PROGRAM prgCS1
VAR
	fbAlfen1					: FB_ECS_Alfen_NG9xx_Platform;						//{#lynus.ag#()}
	fbAlfen2					: FB_ECS_Alfen_NG9xx_Platform;						//{#lynus.ag#()}
	fbAlfen3					: FB_ECS_Alfen_NG9xx_Platform;						//{#lynus.ag#()}
	fbAlfen4					: FB_ECS_Alfen_NG9xx_Platform;						//{#lynus.ag#()}
	fbAlfen5					: FB_ECS_Alfen_NG9xx_Platform;						//{#lynus.ag#()}
	fbAlfen6					: FB_ECS_Alfen_NG9xx_Platform;						//{#lynus.ag#()}
	fbAlfen7					: FB_ECS_Alfen_NG9xx_Platform;						//{#lynus.ag#()}
	fbAlfen8					: FB_ECS_Alfen_NG9xx_Platform;						//{#lynus.ag#()}
	fbAlfen9					: FB_ECS_Alfen_NG9xx_Platform;						//{#lynus.ag#()}
	fbAlfen10					: FB_ECS_Alfen_NG9xx_Platform;						//{#lynus.ag#()}
	fbApliT_1					: FB_ECS_Alpitronic_Hypercharger;					//{#lynus.ag#()}
	fbApliT_2					: FB_ECS_Alpitronic_Hypercharger;					//{#lynus.ag#()}
	
	bSManualyOn_UV1_1			: BOOL;												//{#lynus.ag#()}
	bySManualyTargetPowerUV1_1	: BYTE;												//{#lynus.ag#()}
	byErrorWarningUV1_1			: BYTE;												//{#lynus.ag#()}
	rChargingTimeInMinUV1_1		: REAL;												//{#lynus.ag#()}
	lrPowerUV1_1				: LREAL;											//{#lynus.ag#()}
	wStateUV1_1					: WORD;												//{#lynus.ag#()}
	lrEnergySessionUV1_1		: LREAL;											//{#lynus.ag#()}
	lrTotalEnergyUV1_1			: LREAL;											//{#lynus.ag#()}
	
	bSManualyOn_UV1_2			: BOOL;												//{#lynus.ag#()}
	bySManualyTargetPowerUV1_2	: BYTE;												//{#lynus.ag#()}
	byErrorWarningUV1_2			: BYTE;												//{#lynus.ag#()}
	rChargingTimeInMinUV1_2		: REAL;												//{#lynus.ag#()}
	lrPowerUV1_2				: LREAL;											//{#lynus.ag#()}
	wStateUV1_2					: WORD;												//{#lynus.ag#()}
	lrEnergySessionUV1_2		: LREAL;											//{#lynus.ag#()}
	lrTotalEnergyUV1_2			: LREAL;											//{#lynus.ag#()}
	
	bSManualyOn_UV1_3			: BOOL;												//{#lynus.ag#()}
	bySManualyTargetPowerUV1_3	: BYTE;												//{#lynus.ag#()}
	byErrorWarningUV1_3			: BYTE;												//{#lynus.ag#()}
	rChargingTimeInMinUV1_3		: REAL;												//{#lynus.ag#()}
	lrPowerUV1_3				: LREAL;											//{#lynus.ag#()}
	wStateUV1_3					: WORD;												//{#lynus.ag#()}
	lrEnergySessionUV1_3		: LREAL;											//{#lynus.ag#()}
	lrTotalEnergyUV1_3			: LREAL;											//{#lynus.ag#()}
	
	bSManualyOn_UV1_4			: BOOL;												//{#lynus.ag#()}
	bySManualyTargetPowerUV1_4	: BYTE;												//{#lynus.ag#()}
	byErrorWarningUV1_4			: BYTE;												//{#lynus.ag#()}
	rChargingTimeInMinUV1_4		: REAL;												//{#lynus.ag#()}
	lrPowerUV1_4				: LREAL;											//{#lynus.ag#()}
	wStateUV1_4					: WORD;												//{#lynus.ag#()}
	lrEnergySessionUV1_4		: LREAL;											//{#lynus.ag#()}
	lrTotalEnergyUV1_4			: LREAL;											//{#lynus.ag#()}
	
	bSManualyOn_UV1_5			: BOOL;												//{#lynus.ag#()}
	bySManualyTargetPowerUV1_5	: BYTE;												//{#lynus.ag#()}
	byErrorWarningUV1_5			: BYTE;												//{#lynus.ag#()}
	rChargingTimeInMinUV1_5		: REAL;												//{#lynus.ag#()}
	lrPowerUV1_5				: LREAL;											//{#lynus.ag#()}
	wStateUV1_5					: WORD;												//{#lynus.ag#()}
	lrEnergySessionUV1_5		: LREAL;											//{#lynus.ag#()}
	lrTotalEnergyUV1_5			: LREAL;											//{#lynus.ag#()}
	
	bSManualyOn_UV1_6			: BOOL;												//{#lynus.ag#()}
	bySManualyTargetPowerUV1_6	: BYTE;												//{#lynus.ag#()}
	byErrorWarningUV1_6			: BYTE;												//{#lynus.ag#()}
	rChargingTimeInMinUV1_6		: REAL;												//{#lynus.ag#()}
	lrPowerUV1_6				: LREAL;											//{#lynus.ag#()}
	wStateUV1_6					: WORD;												//{#lynus.ag#()}
	lrEnergySessionUV1_6		: LREAL;											//{#lynus.ag#()}
	lrTotalEnergyUV1_6			: LREAL;											//{#lynus.ag#()}
	
	bSManualyOn_UV1_7			: BOOL;												//{#lynus.ag#()}
	bySManualyTargetPowerUV1_7	: BYTE;												//{#lynus.ag#()}
	byErrorWarningUV1_7			: BYTE;												//{#lynus.ag#()}
	rChargingTimeInMinUV1_7		: REAL;												//{#lynus.ag#()}
	lrPowerUV1_7				: LREAL;											//{#lynus.ag#()}
	wStateUV1_7					: WORD;												//{#lynus.ag#()}
	lrEnergySessionUV1_7		: LREAL;											//{#lynus.ag#()}
	lrTotalEnergyUV1_7			: LREAL;											//{#lynus.ag#()}
	
	bSManualyOn_UV1_8			: BOOL;												//{#lynus.ag#()}
	bySManualyTargetPowerUV1_8	: BYTE;												//{#lynus.ag#()}
	byErrorWarningUV1_8			: BYTE;												//{#lynus.ag#()}
	rChargingTimeInMinUV1_8		: REAL;												//{#lynus.ag#()}
	lrPowerUV1_8				: LREAL;											//{#lynus.ag#()}
	wStateUV1_8					: WORD;												//{#lynus.ag#()}
	lrEnergySessionUV1_8		: LREAL;											//{#lynus.ag#()}
	lrTotalEnergyUV1_8			: LREAL;											//{#lynus.ag#()}
	
	bSManualyOn_UV1_9			: BOOL;												//{#lynus.ag#()}
	bySManualyTargetPowerUV1_9	: BYTE;												//{#lynus.ag#()}
	byErrorWarningUV1_9			: BYTE;												//{#lynus.ag#()}
	rChargingTimeInMinUV1_9		: REAL;												//{#lynus.ag#()}
	lrPowerUV1_9				: LREAL;											//{#lynus.ag#()}
	wStateUV1_9					: WORD;												//{#lynus.ag#()}
	lrEnergySessionUV1_9		: LREAL;											//{#lynus.ag#()}
	lrTotalEnergyUV1_9			: LREAL;											//{#lynus.ag#()}
	
	bSManualyOn_UV1_10			: BOOL;												//{#lynus.ag#()}
	bySManualyTargetPowerUV1_10	: BYTE;												//{#lynus.ag#()}
	byErrorWarningUV1_10		: BYTE;												//{#lynus.ag#()}
	rChargingTimeInMinUV1_10	: REAL;												//{#lynus.ag#()}
	lrPowerUV1_10				: LREAL;											//{#lynus.ag#()}
	wStateUV1_10				: WORD;												//{#lynus.ag#()}
	lrEnergySessionUV1_10		: LREAL;											//{#lynus.ag#()}
	lrTotalEnergyUV1_10			: LREAL;											//{#lynus.ag#()}
	
	bSManualyOn_DC_1			: BOOL;												//{#lynus.ag#()}
	bySManualyTargetPowerDC_1	: BYTE;												//{#lynus.ag#()}
	byErrorWarningDC_1			: BYTE;												//{#lynus.ag#()}
	lrPowerTotalDC1				: LREAL;											//{#lynus.ag#()}
	lrPowerDC1_S1				: LREAL;											//{#lynus.ag#()}
	lrPowerDC1_S2				: LREAL;											//{#lynus.ag#()}
	rChargingTimeInMinDC1_S1	: REAL;												//{#lynus.ag#()}
	rChargingTimeInMinDC1_S2	: REAL;												//{#lynus.ag#()}
	dwSOCCarDC1_S1				: DWORD;											//{#lynus.ag#()}
	dwSOCCarDC1_S2				: DWORD;											//{#lynus.ag#()}
	wStateDC1_S1				: WORD;												//{#lynus.ag#()}
	wStateDC1_S2				: WORD;												//{#lynus.ag#()}
	lrEnergySessionDC1_S1		: LREAL;											//{#lynus.ag#()}
	lrEnergySessionDC1_S2		: LREAL;											//{#lynus.ag#()}
	lrTotalEnergyDC1			: LREAL;											//{#lynus.ag#()}
	
	bSManualyOn_DC_2			: BOOL;												//{#lynus.ag#()}
	bySManualyTargetPowerDC_2	: BYTE;												//{#lynus.ag#()}
	byErrorWarningDC_2			: BYTE;												//{#lynus.ag#()}
	lrPowerTotalDC2				: LREAL;											//{#lynus.ag#()}
	lrPowerDC2_S1				: LREAL;											//{#lynus.ag#()}
	lrPowerDC2_S2				: LREAL;											//{#lynus.ag#()}
	rChargingTimeInMinDC2_S1	: REAL;												//{#lynus.ag#()}
	rChargingTimeInMinDC2_S2	: REAL;												//{#lynus.ag#()}
	dwSOCCarDC2_S1				: DWORD;											//{#lynus.ag#()}
	dwSOCCarDC2_S2				: DWORD;											//{#lynus.ag#()}
	wStateDC2_S1				: WORD;												//{#lynus.ag#()}
	wStateDC2_S2				: WORD;												//{#lynus.ag#()}
	lrEnergySessionDC2_S1		: LREAL;											//{#lynus.ag#()}
	lrEnergySessionDC2_S2		: LREAL;											//{#lynus.ag#()}
	lrTotalEnergyDC2			: LREAL;											//{#lynus.ag#()}
END_VAR
VAR PERSISTENT
	bManualyOnUV1_1				: BOOL;												//{#lynus.ag#()}
	byManualyTargetPowerUV1_1	: BYTE;												//{#lynus.ag#()}
	
	bManualyOnUV1_2				: BOOL;												//{#lynus.ag#()}
	byManualyTargetPowerUV1_2	: BYTE;												//{#lynus.ag#()}
	
	bManualyOnUV1_3				: BOOL;												//{#lynus.ag#()}
	byManualyTargetPowerUV1_3	: BYTE;												//{#lynus.ag#()}
	
	bManualyOnUV1_4				: BOOL;												//{#lynus.ag#()}
	byManualyTargetPowerUV1_4	: BYTE;												//{#lynus.ag#()}
	
	bManualyOnUV1_5				: BOOL;												//{#lynus.ag#()}
	byManualyTargetPowerUV1_5	: BYTE;												//{#lynus.ag#()}
	
	bManualyOnUV1_6				: BOOL;												//{#lynus.ag#()}
	byManualyTargetPowerUV1_6	: BYTE;												//{#lynus.ag#()}
	
	bManualyOnUV1_7				: BOOL;												//{#lynus.ag#()}
	byManualyTargetPowerUV1_7	: BYTE;												//{#lynus.ag#()}
	
	bManualyOnUV1_8				: BOOL;												//{#lynus.ag#()}
	byManualyTargetPowerUV1_8	: BYTE;												//{#lynus.ag#()}
	
	bManualyOnUV1_9				: BOOL;												//{#lynus.ag#()}
	byManualyTargetPowerUV1_9	: BYTE;												//{#lynus.ag#()}
	
	bManualyOnUV1_10			: BOOL;												//{#lynus.ag#()}
	byManualyTargetPowerUV1_10	: BYTE;												//{#lynus.ag#()}
	
	bManualyOnDC_1				: BOOL;												//{#lynus.ag#()}
	byManualyTargetPowerDC_1	: BYTE;												//{#lynus.ag#()}
	
	bManualyOnDC_2				: BOOL;												//{#lynus.ag#()}
	byManualyTargetPowerDC_2	: BYTE;												//{#lynus.ag#()}
END_VAR

(*---------------------------------------------CS1-----------------------------------------------------------*)

//Manual Power
fbAlfen1.stSetupECS.bManualyOn := bManualyOnUV1_1;
	fbAlfen1.stSetupECS.byManualyTargetPower := byManualyTargetPowerUV1_1;

fbAlfen1(
	bEnable:= , 
	bPowerDataInvers:= , 
	byElectricFuseLine:= , 
	byUnitID_Socket1:= 1, 
	byUnitID_Socket2:= , 
	byNumberOfSockets:= 1, 
	byNumberOfConnectionWire:= 1, 
	diNrOfEMS_IN:= prgEMS.fbEMS.diNrOfEMS_OUT, 
	diNrOfEM_IN_CS:= , 
	sIPAdress:= '192.168.1.123', 
	stSetupECS:= , 
	stDataECS=> , 
	diNrOfECS_OUT=> );

bSManualyOn_UV1_1 := fbAlfen1.stDataECS.bSManualyOn;
	bySManualyTargetPowerUV1_1 := fbAlfen1.stDataECS.bySManualyTargetPower;
		byErrorWarningUV1_1 := fbAlfen1.stDataECS.byErrorWarning;	
			rChargingTimeInMinUV1_1 := fbAlfen1.stDataECS.arrChargingTimeInMin[1];
				lrPowerUV1_1 := fbAlfen1.stDataECS.lrTotalPower;	
					wStateUV1_1 := fbAlfen1.stDataECS.arrSocketStateECS[1];
						lrEnergySessionUV1_1 := fbAlfen1.stDataECS.arrSocketEnergySession[1];
							lrTotalEnergyUV1_1 := fbAlfen1.stDataECS.lrTotalCounterEnergy_Consumption;		
	
(*---------------------------------------------CS2-----------------------------------------------------------*)
	
//Manual Power
fbAlfen2.stSetupECS.bManualyOn := bManualyOnUV1_2;
	fbAlfen2.stSetupECS.byManualyTargetPower := byManualyTargetPowerUV1_2;
	
fbAlfen2(
	bEnable:= , 
	bPowerDataInvers:= , 
	byElectricFuseLine:= , 
	byUnitID_Socket1:= 1, 
	byUnitID_Socket2:= , 
	byNumberOfSockets:= 1, 
	byNumberOfConnectionWire:= 1, 
	diNrOfEMS_IN:= prgEMS.fbEMS.diNrOfEMS_OUT, 
	diNrOfEM_IN_CS:= , 
	sIPAdress:= '192.168.1.111', 
	stSetupECS:= , 
	stDataECS=> , 
	diNrOfECS_OUT=> );

bSManualyOn_UV1_2 := fbAlfen2.stDataECS.bSManualyOn;
	bySManualyTargetPowerUV1_2 := fbAlfen2.stDataECS.bySManualyTargetPower;	
		byErrorWarningUV1_2 := fbAlfen2.stDataECS.byErrorWarning;
			rChargingTimeInMinUV1_2 := fbAlfen2.stDataECS.arrChargingTimeInMin[1];;
				lrPowerUV1_2 := fbAlfen2.stDataECS.lrTotalPower;	
					wStateUV1_2 := fbAlfen2.stDataECS.arrSocketStateECS[1];
						lrEnergySessionUV1_2 := fbAlfen2.stDataECS.arrSocketEnergySession[1];
							lrTotalEnergyUV1_2 := fbAlfen2.stDataECS.lrTotalCounterEnergy_Consumption;
	
(*---------------------------------------------CS3-----------------------------------------------------------*)	
	
//Manual Power
fbAlfen3.stSetupECS.bManualyOn := bManualyOnUV1_3;
	fbAlfen3.stSetupECS.byManualyTargetPower := byManualyTargetPowerUV1_3;
	
fbAlfen3(
	bEnable:= , 
	bPowerDataInvers:= , 
	byElectricFuseLine:= , 
	byUnitID_Socket1:= 1, 
	byUnitID_Socket2:= , 
	byNumberOfSockets:= 1, 
	byNumberOfConnectionWire:= 1, 
	diNrOfEMS_IN:= prgEMS.fbEMS.diNrOfEMS_OUT, 
	diNrOfEM_IN_CS:= , 
	sIPAdress:= '192.168.1.213',  
	stSetupECS:= , 
	stDataECS=> , 
	diNrOfECS_OUT=> );

bSManualyOn_UV1_3 := fbAlfen3.stDataECS.bSManualyOn;
	bySManualyTargetPowerUV1_3 := fbAlfen3.stDataECS.bySManualyTargetPower;
		byErrorWarningUV1_3 := fbAlfen3.stDataECS.byErrorWarning;
			rChargingTimeInMinUV1_3 := fbAlfen3.stDataECS.arrChargingTimeInMin[1];	
				lrPowerUV1_3 := fbAlfen3.stDataECS.lrTotalPower;	
					wStateUV1_3 := fbAlfen3.stDataECS.arrSocketStateECS[1];
						lrEnergySessionUV1_3 := fbAlfen3.stDataECS.arrSocketEnergySession[1];
							lrTotalEnergyUV1_3 := fbAlfen3.stDataECS.lrTotalCounterEnergy_Consumption;
	
(*---------------------------------------------CS4-----------------------------------------------------------*)	
	
//Manual Power
fbAlfen4.stSetupECS.bManualyOn := bManualyOnUV1_4;
	fbAlfen4.stSetupECS.byManualyTargetPower := byManualyTargetPowerUV1_4;
	
fbAlfen4(
	bEnable:= , 
	bPowerDataInvers:= , 
	byElectricFuseLine:= , 
	byUnitID_Socket1:= 1, 
	byUnitID_Socket2:= , 
	byNumberOfSockets:= 1, 
	byNumberOfConnectionWire:= 1, 
	diNrOfEMS_IN:= prgEMS.fbEMS.diNrOfEMS_OUT, 
	diNrOfEM_IN_CS:= , 
	sIPAdress:= '192.168.1.144',  
	stSetupECS:= , 
	stDataECS=> , 
	diNrOfECS_OUT=> );

bSManualyOn_UV1_4 := fbAlfen4.stDataECS.bSManualyOn;
	bySManualyTargetPowerUV1_4 := fbAlfen4.stDataECS.bySManualyTargetPower;	
		byErrorWarningUV1_4 := fbAlfen4.stDataECS.byErrorWarning;
			rChargingTimeInMinUV1_4 := fbAlfen4.stDataECS.arrChargingTimeInMin[1];
				lrPowerUV1_4 := fbAlfen4.stDataECS.lrTotalPower;	
					wStateUV1_4 := fbAlfen4.stDataECS.arrSocketStateECS[1];
						lrEnergySessionUV1_4 := fbAlfen4.stDataECS.arrSocketEnergySession[1];
							lrTotalEnergyUV1_4 := fbAlfen4.stDataECS.lrTotalCounterEnergy_Consumption;
	
(*---------------------------------------------CS5-----------------------------------------------------------*)	
	
//Manual Power
fbAlfen5.stSetupECS.bManualyOn := bManualyOnUV1_5;
	fbAlfen5.stSetupECS.byManualyTargetPower := byManualyTargetPowerUV1_5;
	
fbAlfen5(
	bEnable:= , 
	bPowerDataInvers:= , 
	byElectricFuseLine:= , 
	byUnitID_Socket1:= 1, 
	byUnitID_Socket2:= , 
	byNumberOfSockets:= 1, 
	byNumberOfConnectionWire:= 1, 
	diNrOfEMS_IN:= prgEMS.fbEMS.diNrOfEMS_OUT, 
	diNrOfEM_IN_CS:= , 
	sIPAdress:= '192.168.1.178',  
	stSetupECS:= , 
	stDataECS=> , 
	diNrOfECS_OUT=> );

bSManualyOn_UV1_5 := fbAlfen5.stDataECS.bSManualyOn;
	bySManualyTargetPowerUV1_5 := fbAlfen5.stDataECS.bySManualyTargetPower;
		byErrorWarningUV1_5 := fbAlfen5.stDataECS.byErrorWarning;
			rChargingTimeInMinUV1_5 := fbAlfen5.stDataECS.arrChargingTimeInMin[1];
				lrPowerUV1_5 := fbAlfen5.stDataECS.lrTotalPower;	
					wStateUV1_5 := fbAlfen5.stDataECS.arrSocketStateECS[1];
						lrEnergySessionUV1_5 := fbAlfen5.stDataECS.arrSocketEnergySession[1];
							lrTotalEnergyUV1_5 := fbAlfen5.stDataECS.lrTotalCounterEnergy_Consumption;	
	
(*---------------------------------------------CS6-----------------------------------------------------------*)	
	
//Manual Power
fbAlfen6.stSetupECS.bManualyOn := bManualyOnUV1_6;
	fbAlfen6.stSetupECS.byManualyTargetPower := byManualyTargetPowerUV1_6;
	
fbAlfen6(
	bEnable:= , 
	bPowerDataInvers:= , 
	byElectricFuseLine:= , 
	byUnitID_Socket1:= 1, 
	byUnitID_Socket2:= , 
	byNumberOfSockets:= 1, 
	byNumberOfConnectionWire:= 1, 
	diNrOfEMS_IN:= prgEMS.fbEMS.diNrOfEMS_OUT, 
	diNrOfEM_IN_CS:= , 
	sIPAdress:= '192.168.1.161',  
	stSetupECS:= , 
	stDataECS=> , 
	diNrOfECS_OUT=> );

bSManualyOn_UV1_6 := fbAlfen6.stDataECS.bSManualyOn;
	bySManualyTargetPowerUV1_6 := fbAlfen6.stDataECS.bySManualyTargetPower;	
		byErrorWarningUV1_6 := fbAlfen6.stDataECS.byErrorWarning;
			rChargingTimeInMinUV1_6 := fbAlfen6.stDataECS.arrChargingTimeInMin[1];
				lrPowerUV1_6 := fbAlfen6.stDataECS.lrTotalPower;	
					wStateUV1_6 := fbAlfen6.stDataECS.arrSocketStateECS[1];
						lrEnergySessionUV1_6 := fbAlfen6.stDataECS.arrSocketEnergySession[1];
							lrTotalEnergyUV1_6 := fbAlfen6.stDataECS.lrTotalCounterEnergy_Consumption;
	
(*---------------------------------------------CS7-----------------------------------------------------------*)	
	
//Manual Power
fbAlfen7.stSetupECS.bManualyOn := bManualyOnUV1_7;
	fbAlfen7.stSetupECS.byManualyTargetPower := byManualyTargetPowerUV1_7;
	
fbAlfen7(
	bEnable:= , 
	bPowerDataInvers:= , 
	byElectricFuseLine:= , 
	byUnitID_Socket1:= 1, 
	byUnitID_Socket2:= , 
	byNumberOfSockets:= 1, 
	byNumberOfConnectionWire:= 1, 
	diNrOfEMS_IN:= prgEMS.fbEMS.diNrOfEMS_OUT, 
	diNrOfEM_IN_CS:= , 
	sIPAdress:= '192.168.1.241',  
	stSetupECS:= , 
	stDataECS=> , 
	diNrOfECS_OUT=> );

bSManualyOn_UV1_7 := fbAlfen7.stDataECS.bSManualyOn;
	bySManualyTargetPowerUV1_7 := fbAlfen7.stDataECS.bySManualyTargetPower;	
		byErrorWarningUV1_7 := fbAlfen7.stDataECS.byErrorWarning;
			rChargingTimeInMinUV1_7 := fbAlfen7.stDataECS.arrChargingTimeInMin[1];
				lrPowerUV1_7 := fbAlfen7.stDataECS.lrTotalPower;	
					wStateUV1_7 := fbAlfen7.stDataECS.arrSocketStateECS[1];
						lrEnergySessionUV1_7 := fbAlfen7.stDataECS.arrSocketEnergySession[1];
							lrTotalEnergyUV1_7 := fbAlfen7.stDataECS.lrTotalCounterEnergy_Consumption;
	
(*---------------------------------------------CS8-----------------------------------------------------------*)	
	
//Manual Power
fbAlfen8.stSetupECS.bManualyOn := bManualyOnUV1_8;
	fbAlfen8.stSetupECS.byManualyTargetPower := byManualyTargetPowerUV1_8;
	
fbAlfen8(
	bEnable:= , 
	bPowerDataInvers:= , 
	byElectricFuseLine:= , 
	byUnitID_Socket1:= 1, 
	byUnitID_Socket2:= , 
	byNumberOfSockets:= 1, 
	byNumberOfConnectionWire:= 1, 
	diNrOfEMS_IN:= prgEMS.fbEMS.diNrOfEMS_OUT, 
	diNrOfEM_IN_CS:= , 
	sIPAdress:= '192.168.1.124',  
	stSetupECS:= , 
	stDataECS=> , 
	diNrOfECS_OUT=> );

bSManualyOn_UV1_8 := fbAlfen8.stDataECS.bSManualyOn;
	bySManualyTargetPowerUV1_8 := fbAlfen8.stDataECS.bySManualyTargetPower;	
		byErrorWarningUV1_8 := fbAlfen8.stDataECS.byErrorWarning;
			rChargingTimeInMinUV1_8 := fbAlfen8.stDataECS.arrChargingTimeInMin[1];
				lrPowerUV1_8 := fbAlfen8.stDataECS.lrTotalPower;	
					wStateUV1_8 := fbAlfen8.stDataECS.arrSocketStateECS[1];
						lrEnergySessionUV1_8 := fbAlfen8.stDataECS.arrSocketEnergySession[1];
							lrTotalEnergyUV1_8 := fbAlfen8.stDataECS.lrTotalCounterEnergy_Consumption;
	
(*---------------------------------------------CS9-----------------------------------------------------------*)	
	
//Manual Power
fbAlfen9.stSetupECS.bManualyOn := bManualyOnUV1_9;
	fbAlfen9.stSetupECS.byManualyTargetPower := byManualyTargetPowerUV1_9;
	
fbAlfen9(
	bEnable:= , 
	bPowerDataInvers:= , 
	byElectricFuseLine:= , 
	byUnitID_Socket1:= 1, 
	byUnitID_Socket2:= , 
	byNumberOfSockets:= 1, 
	byNumberOfConnectionWire:= 1, 
	diNrOfEMS_IN:= prgEMS.fbEMS.diNrOfEMS_OUT, 
	diNrOfEM_IN_CS:= , 
	sIPAdress:= '192.168.1.165',  
	stSetupECS:= , 
	stDataECS=> , 
	diNrOfECS_OUT=> );

bSManualyOn_UV1_9 := fbAlfen9.stDataECS.bSManualyOn;
	bySManualyTargetPowerUV1_9 := fbAlfen9.stDataECS.bySManualyTargetPower;
		byErrorWarningUV1_9 := fbAlfen9.stDataECS.byErrorWarning;	
			rChargingTimeInMinUV1_9 := fbAlfen9.stDataECS.arrChargingTimeInMin[1];
				lrPowerUV1_9 := fbAlfen9.stDataECS.lrTotalPower;	
					wStateUV1_9 := fbAlfen9.stDataECS.arrSocketStateECS[1];
						lrEnergySessionUV1_9 := fbAlfen9.stDataECS.arrSocketEnergySession[1];
							lrTotalEnergyUV1_9 := fbAlfen9.stDataECS.lrTotalCounterEnergy_Consumption;
	
(*---------------------------------------------CS10-----------------------------------------------------------*)	
	
//Manual Power
fbAlfen10.stSetupECS.bManualyOn := bManualyOnUV1_10;
	fbAlfen10.stSetupECS.byManualyTargetPower := byManualyTargetPowerUV1_10;
	
fbAlfen10(
	bEnable:= , 
	bPowerDataInvers:= , 
	byElectricFuseLine:= , 
	byUnitID_Socket1:= 1, 
	byUnitID_Socket2:= , 
	byNumberOfSockets:= 1, 
	byNumberOfConnectionWire:= 1, 
	diNrOfEMS_IN:= prgEMS.fbEMS.diNrOfEMS_OUT, 
	diNrOfEM_IN_CS:= , 
	sIPAdress:= '192.168.1.176', 
	stSetupECS:= , 
	stDataECS=> , 
	diNrOfECS_OUT=> );

bSManualyOn_UV1_10 := fbAlfen10.stDataECS.bSManualyOn;
	bySManualyTargetPowerUV1_10 := fbAlfen10.stDataECS.bySManualyTargetPower;
		byErrorWarningUV1_10 := fbAlfen10.stDataECS.byErrorWarning;	
			rChargingTimeInMinUV1_10 := fbAlfen10.stDataECS.arrChargingTimeInMin[1];
				lrPowerUV1_10 := fbAlfen10.stDataECS.lrTotalPower;	
					wStateUV1_10 := fbAlfen10.stDataECS.arrSocketStateECS[1];
						lrEnergySessionUV1_10 := fbAlfen10.stDataECS.arrSocketEnergySession[1];
							lrTotalEnergyUV1_10 := fbAlfen10.stDataECS.lrTotalCounterEnergy_Consumption;

(*---------------------------------------------DC1-----------------------------------------------------------*)	
	
//Manual Power
fbApliT_1.stSetupECS.bManualyOn := bManualyOnDC_1;
	fbApliT_1.stSetupECS.byManualyTargetPower := byManualyTargetPowerDC_1;
	
fbApliT_1(
	bEnable:= , 
	bPowerDataInvers:= , 
	byElectricFuseLine:= , 
	byUnitID:= 1, 
	diNrOfEMS_IN:= prgEMS.fbEMS.diNrOfEMS_OUT, 
	diNrOfEM_IN_CS:= , 
	sIPAdress:= '192.168.1.177', 
	stSetupECS:= , 
	stDataECS=> , 
	diNrOfECS_OUT=> );

bSManualyOn_DC_1 := fbApliT_1.stDataECS.bSManualyOn;
	bySManualyTargetPowerDC_1 := fbApliT_1.stDataECS.bySManualyTargetPower;
		byErrorWarningDC_1 := fbApliT_1.stDataECS.byErrorWarning;
			lrPowerTotalDC1 := fbApliT_1.stDataECS.lrTotalPower;
				lrPowerDC1_S1 :=  fbApliT_1.stDataECS.arrSocketPower[1];
					lrPowerDC1_S2 :=  fbApliT_1.stDataECS.arrSocketPower[2];	 	
						rChargingTimeInMinDC1_S1 := fbApliT_1.stDataECS.arrChargingTimeInMin[1];	
							rChargingTimeInMinDC1_S2 := fbApliT_1.stDataECS.arrChargingTimeInMin[2];
								dwSOCCarDC1_S1 := fbApliT_1.stDataECS.arrSocketSOCCar[1]; 
									dwSOCCarDC1_S2 := fbApliT_1.stDataECS.arrSocketSOCCar[2]; 	
										wStateDC1_S1 := fbApliT_1.stDataECS.arrSocketStateECS[1];
											wStateDC1_S2 := fbApliT_1.stDataECS.arrSocketStateECS[2];
												lrEnergySessionDC1_S1 := fbApliT_1.stDataECS.arrSocketEnergySession[1];
													lrEnergySessionDC1_S2 := fbApliT_1.stDataECS.arrSocketEnergySession[2];
														lrTotalEnergyDC1 := fbApliT_1.stDataECS.lrTotalCounterEnergy_Consumption;			
		
(*---------------------------------------------DC2-----------------------------------------------------------*)	
	
//Manual Power
fbApliT_2.stSetupECS.bManualyOn := bManualyOnDC_2;
	fbApliT_2.stSetupECS.byManualyTargetPower := byManualyTargetPowerDC_2;
	
fbApliT_2(
	bEnable:= , 
	bPowerDataInvers:= , 
	byElectricFuseLine:= , 
	byUnitID:= 1, 
	diNrOfEMS_IN:= prgEMS.fbEMS.diNrOfEMS_OUT, 
	diNrOfEM_IN_CS:= , 
	sIPAdress:= '192.168.1.185', 
	stSetupECS:= , 
	stDataECS=> , 
	diNrOfECS_OUT=> );
	
bSManualyOn_DC_2 := fbApliT_2.stDataECS.bSManualyOn;
	bySManualyTargetPowerDC_2 := fbApliT_2.stDataECS.bySManualyTargetPower;
		byErrorWarningDC_2 := fbApliT_2.stDataECS.byErrorWarning;
			lrPowerTotalDC2 := fbApliT_2.stDataECS.lrTotalPower;
				lrPowerDC2_S1 :=  fbApliT_2.stDataECS.arrSocketPower[1];
					lrPowerDC2_S2 :=  fbApliT_2.stDataECS.arrSocketPower[2];	 	
						rChargingTimeInMinDC2_S1 := fbApliT_2.stDataECS.arrChargingTimeInMin[1];	
							rChargingTimeInMinDC2_S2 := fbApliT_2.stDataECS.arrChargingTimeInMin[2];
								dwSOCCarDC2_S1 := fbApliT_2.stDataECS.arrSocketSOCCar[1]; 
									dwSOCCarDC2_S2 := fbApliT_2.stDataECS.arrSocketSOCCar[2]; 	
										wStateDC2_S1 := fbApliT_2.stDataECS.arrSocketStateECS[1];
											wStateDC2_S2 := fbApliT_2.stDataECS.arrSocketStateECS[2];
												lrEnergySessionDC2_S1 := fbApliT_2.stDataECS.arrSocketEnergySession[1];
													lrEnergySessionDC2_S2 := fbApliT_2.stDataECS.arrSocketEnergySession[2];
														lrTotalEnergyDC2 := fbApliT_2.stDataECS.lrTotalCounterEnergy_Consumption;

END_PROGRAM

(* stored: Version 1.1.0.1, ProductVersion 3.1.4024.9
   POU prgCS1: Id {73274ddf-8b0e-46f2-b052-ab4c1bcb19dd}, SpecialFunc None *)
